// TIA Portal V21 export
VAR_GLOBAL   // PLC tag table "DO"
   "VCC PUMP" AT %Q0.0 : Bool;   // VCC PUMP
   "DOOR1 GASKET" AT %Q0.1 : Bool;   // DOOR1 GASKET
   "DOOR1 VCC" AT %Q0.2 : Bool;   // DOOR1 VCC
   "DOOR2 GASKET" AT %Q0.3 : Bool;   // DOOR2 GASKET
   "DOOR2 VCC" AT %Q0.4 : Bool;   // DOOR2 VCC
   "JACKET STEAM VAL" AT %Q0.5 : Bool;   // JACKET STEAM VAL
   "JACKET STEAM OUT" AT %Q0.6 : Bool;
   "CHAMBER STEAM VAL" AT %Q0.7 : Bool;   // CHAMBER STEAM VAL
   "CHAMBER STEAM SMALL" AT %Q1.0 : Bool;   // DOOR2 INTERLOCK VAL
   "CHAMBER EXHAUST VAL" AT %Q1.1 : Bool;   // CHAMBER EXHAUST VAL
   "DRAIN VAL" AT %Q2.0 : Bool;   // DRAIN VAL
   "CHAMBER VACCUM VAL" AT %Q2.1 : Bool;
   "CHAMBER VENT VAL" AT %Q2.2 : Bool;   // CHAMBER VENT VAL
   "DOOR1 OPEN VAL" AT %Q2.3 : Bool;   // DOOR1 OPEN VAL
   "DOOR1 CLOSE VAL" AT %Q2.4 : Bool;   // DOOR1 CLOSE VAL
   "DOOR2 OPEN VAL" AT %Q2.5 : Bool;   // DOOR2 OPEN VAL
   "DOOR2 CLOSE VAL" AT %Q2.6 : Bool;   // DOOR2 CLOSE VAL
   "PROCESS ON IND" AT %Q2.7 : Bool;   // WFI VAL
   "door1 precondition lamp" AT %Q3.0 : Bool;
   "door2 precondition lamp" AT %Q3.1 : Bool;
   "DOOR1 OPEN LAMP" AT %Q3.2 : Bool;   // PWD VAL
   "DOOR2 OPEN LAMP" AT %Q3.3 : Bool;   // PWD CRC VAL
   HOOTER AT %Q3.4 : Bool;   // HOOTER
   "CHAMBER CONDENSOR VAL" AT %Q3.5 : Bool;   // CHAMBER CONDENSOR VAL
   "BOILER HEATER" AT %Q3.6 : Bool;   // BOILER HEATER
   "CRC MOTOR" AT %Q10.2 : Bool;   // CRC MOTOR
   "DETERGENT DSG VAL" AT %Q12.2 : Bool;   // DETERGENT DSG VAL
   "SILICON DSG VAL" AT %Q12.3 : Bool;   // SILICON DSG VAL
   "CHAMBER AIR VENT FAST" AT %Q18.6 : Bool;   // DOOR1 INTERLOCK VAL
END_VAR
